// TIA Portal V17 export
// export: Created 2021-12-03T08:12:55.8900869Z, ExportSetting WithDefaults, DisplayName Totally Integrated Automation Portal, DisplayVersion V17, DisplayName TIA Portal Openness, DisplayVersion V17, DisplayName TIA Portal Version Control Interface, DisplayVersion V17, DisplayName STEP 7 Professional, DisplayVersion V17, DisplayName STEP 7 Safety, DisplayVersion V17, DisplayName WinCC Advanced, DisplayVersion V17
DATA_BLOCK "DBI_DetLineSts"   // DB25
VERSION : 0.1
// stored: AutoNumber false, InstanceOfName FB_DetLineSts, InstanceOfType FB
"FB_DetLineSts"
   // VAR_INPUT
   //    ID { ExternalVisible := 'False'} : Int;
   //    LADDR { ExternalVisible := 'False'} : Word;
   //    I_FltAck { ExternalVisible := 'False'} : Bool;
   // END_VAR
   // VAR_OUTPUT
   //    O_ConOk { ExternalVisible := 'False'; ExternalWritable := 'False'} : Bool;
   //    O_SyncStrt { ExternalVisible := 'False'; ExternalWritable := 'False'} : Bool;
   //    O_ScanAct { ExternalVisible := 'False'; ExternalWritable := 'False'} : Bool;
   //    O_RdyForScan { ExternalVisible := 'False'; ExternalWritable := 'False'} : Bool;
   //    O_ErrRdyAck { ExternalVisible := 'False'; ExternalWritable := 'False'} : Bool;
   //    O_State { ExternalVisible := 'False'; ExternalWritable := 'False'} : Int;
   //    O_ErgMd { ExternalVisible := 'False'; ExternalWritable := 'False'} : Int;
   //    O_TrigRate { ExternalVisible := 'False'; ExternalWritable := 'False'} : Int;
   // END_VAR
   // VAR RETAIN
   //    DetLine_Sts { ExternalVisible := 'False'; ExternalWritable := 'False'} : Struct
   //       MsgId { ExternalVisible := 'False'; ExternalWritable := 'False'} : DWord;
   //       MsgLen { ExternalVisible := 'False'; ExternalWritable := 'False'} : DWord;
   //       Sts { ExternalVisible := 'False'; ExternalWritable := 'False'} : DWord;
   //       State { ExternalVisible := 'False'; ExternalWritable := 'False'} : DWord;
   //       ErgMode { ExternalVisible := 'False'; ExternalWritable := 'False'} : DWord;
   //       TrigRate { ExternalVisible := 'False'; ExternalWritable := 'False'} : DWord;
   //    END_STRUCT;
   //    TCP_Sts { ExternalVisible := 'False'} : Struct
   //       Done { ExternalVisible := 'False'} : Bool;
   //       Error { ExternalVisible := 'False'} : Bool;
   //       Status { ExternalVisible := 'False'} : Word;
   //       Len { ExternalVisible := 'False'} : Int;
   //       ErrCd { ExternalVisible := 'False'} : Word;
   //    END_STRUCT;
   //    AxPtrig { ExternalVisible := 'False'} : Struct
   //       Done { ExternalVisible := 'False'} : Bool;
   //    END_STRUCT;
   //    S_AckRq { ExternalVisible := 'False'} : Bool;
   //    S_Con_Nok { ExternalVisible := 'False'} : Bool;
   // END_VAR
BEGIN
END_DATA_BLOCK
